(* PLC project  *)

CONFIGURATION Robot_B
END_CONFIGURATION
